VAR_GLOBAL PERSISTENT
	G_xExistCAxis:					BOOL:=TRUE;							//TRUE:=Exist C-Axis, FALSE:=Not exist C-Axis
	G_xComProtocol:					BOOL:= TRUE;						//TRUE:=OPC, FALSE:=LOCAL
	//Individual axis positions like fider position...
	G_asIndividualAxisPositions:		ARRAY [1..CE_AXIS_C] OF tsAxisPositions;
	//Min/Max/Offset parameters for drives...
	G_asDriveParameters:				ARRAY [1..CE_AXIS_C] OF tsDriveParameter:= [(PositionMin:=-40.00,	PositionMax:=640.00,		PositionOffset:=-293.00),	(*X-Axis initial parameters*)
																					(PositionMin:=-193.00,	PositionMax:=530.00,	PositionOffset:=240.00),	(*Y-Axis initial parameters*)
																					(PositionMin:=-3,		PositionMax:=252,		PositionOffset:=127.00), 	(*Z-Axis initial parameters*)
																					(PositionMin:=0,		PositionMax:=0,			PositionOffset:=0.00)];		(*C-Axis initial parameters*)
		
END_VAR

(* stored: Version 1.1.0.1, ProductVersion 3.1.4022.18
   GVL PERSIST_GLV: Id {d47ccd71-0f2e-45fa-bb9b-384e297f704f} *)
